# EPICS autosave request: support/areaDetector-s55/iocBoot/iocPVCam/auto_settings.req
file "pvCam_settings.req",  	  P=$(P),  R=pvcam:
file "ADBase_settings.req",       P=$(P),  R=pvcam:
file "NDPluginBase_settings.req", P=$(P),  R=image:
file "NDStdArrays_settings.req",  P=$(P),  R=image:
file "commonPlugin_settings.req", P=$(P)
